FUNCTION_BLOCK FB_TrackSegment_1 EXTENDS FB_TrackBase IMPLEMENTS I_TRACK
VAR_INPUT
END_VAR
VAR_OUTPUT
END_VAR

METHOD Initialize : BOOL
VAR_INPUT
	nTrackIndex : UDINT;
END_VAR

VAR_INST
	TrackTable		: FB_TrackTable;
	
	nPointIndex		: INT;
	nPointIndexA	: INT;	
	nPointIndexB	: INT;	
	idx1, idx2		: INT;
	nStartFromTrack	: INT;
	nEndAtTrack		: INT;
	bCloseLoop		: BOOL;	
	
	bTrackBuild		: BOOL;
	StartFromTrack	: I_Track;
	EndAtTrack		: I_Track;
	
	sIndexWhereTheCheckFailed	: UINT;
	nErrorID					: UDINT;

END_VAR





VAR_INST
	
	TrackTableTemp		: ARRAY[1..gc_MaxNumberTrackPoints] OF ST_TrackTable;
	


END_VAR


VAR_INST
	
	pos01	:		PositionXYC;
	pos02	:		PositionXYC;


END_VAR

	  
CASE nState OF 

	10:	// Starting with an empty table. 
		IF TrackTable.ClearTrackTable() THEN
			nState := nState + 10;
		END_IF
		

	20:	// Init Track-Table
		
		// *************************************************************************************
		// *** Only the code in this state must be eddited according to machine/track layout ***
		// *************************************************************************************	
		
		nStartFromTrack	:= 0;		// 0 for the first track all others according to their predecessor!
	    	nEndAtTrack := 0;		// 0 for the first track all others according to their successor! 		
		     bCloseLoop := FALSE;	// TRUE for circular track	

			 			 			 
		// Building the track table:	
		TrackTable.AddPoint(E_PointType.Line_Start, E_PointOption.none, 480.0, 120.0, 0.0); 	 
		TrackTable.AddPoint(E_PointType.Line_End,   E_PointOption.none, 240.0, 120.0, 0.0);				
		
		TrackTable.AddPoint(E_PointType.Line_Start, E_PointOption.none, 120.0, 240.0, 0.0); 	 
		TrackTable.AddPoint(E_PointType.Line_End,   E_PointOption.none, 120.0, 480.0, 0.0);	
 
		TrackTable.AddPoint(E_PointType.Line_Start, E_PointOption.none, 240.0, 600.0, 0.0); 	 
		TrackTable.AddPoint(E_PointType.Line_End,   E_PointOption.none, 480.0, 600.0, 0.0);		
	 		
		nState := nState + 10;


	30:
		// *************************************************************
		// ***       NO Code Changes are needed from here on!        ***
		// *************************************************************		
			
		// The track table contains all additional information, too.
		IF nStartFromTrack > 0 THEN
			TrackTable.P_StartFromTrack := ipTrack[nStartFromTrack].std;	
		END_IF
		IF nEndAtTrack > 0 THEN
			TrackTable.P_EndAtTrack := ipTrack[nEndAtTrack].std;	
		END_IF	
		TrackTable.P_CloseTheLoop := bCloseLoop;	
		nState := nState + 10;

			
		
	40: // Checking the track table for plausibility
		IF TrackTable.CheckTrackTable() <> 0 THEN
			IF TrackTable.P_TrackTableCheckResult THEN
				nState := 50;	// Plausibility test succeeded.
			ELSE
				nState := 41;	// Plausibility test failed!
			END_IF
		END_IF

	
	41:	// In case of failed plausibility test check the creation of the above track table.
		// A Line must always begin with E_PointType.Line_Start and end with E_PointType.Line_End.
		// A Circle must always be added in the order E_PointType.Circle_Start, E_PointType.Circle_Center, E_PointType.Circle_End.
		// Check the info text for further information:
		sErrorInfoTextTemp := CONCAT('Track: ', UDINT_TO_STRING(nTrackIndex));
		sErrorInfoTextTemp := CONCAT(sErrorInfoTextTemp, ' - ');
		sErrorInfoTextTemp := CONCAT(sErrorInfoTextTemp, TrackTable.P_InfoText);
		
				     bTrackBuildError := TRUE;
					   sErrorInfoText := sErrorInfoTextTemp;
			sIndexWhereTheCheckFailed := TrackTable.P_TrackCheckImplausibleTableIndex;
					   TrackTableTemp := TrackTable.P_Table;	
							
 					   
	50:	// Building the track	
		IF fbTrackStandard.BuildTrackExt(TrackTable) THEN
			nState := nState +1;
		END_IF
		
	51:	IF fbTrackStandard.P_BuildTrackExt.Done THEN
			nState := 100;	
		ELSIF fbTrackStandard.P_BuildTrackExt.Error THEN
	  		nState := nState +1;
		END_IF		
		
	52: // In case an error occured, check the error ID and InfoText and react accordingly:
		sErrorInfoTextTemp := CONCAT('Track: ', UDINT_TO_STRING(nTrackIndex));
		sErrorInfoTextTemp := CONCAT(sErrorInfoTextTemp, ' - ');
		sErrorInfoTextTemp := CONCAT(sErrorInfoTextTemp, fbTrackStandard.P_BuildTrackExtInfoText);	
	
			      nErrorID := fbTrackStandard.P_BuildTrackExt.ErrorID;
		    sErrorInfoText := sErrorInfoTextTemp;		
			
		  bTrackBuildError := TRUE;		   
					   
		 
	100: 	// Track build done
			fTrackLength := fbTrackStandard.GetLength();
			  Initialize := TRUE;
	

END_CASE
END_METHOD

PROPERTY P_Error : BOOL
GET
P_Error := bTrackBuildError;
END_GET
END_PROPERTY

PROPERTY P_ErrorInfo : STRING
GET
P_ErrorInfo := sErrorInfoText;
END_GET
END_PROPERTY

END_FUNCTION_BLOCK

(* stored: Version 1.1.0.1, ProductVersion 3.1.4024.13
   POU FB_TrackSegment_1: Id {8bc03b03-a8a0-4837-bf56-60fab90a5b15}, SpecialFunc None
   Method Initialize: Id {ec4a5bb1-839f-4f43-b542-fc56fd640856}
   Property P_Error: Id {d386063a-b1d4-4b3c-940b-ef6404cff1d0}
   Get Get: Id {e4cd3f32-fa4c-420e-b6e4-48cb575ffb24}
   Property P_ErrorInfo: Id {1e4f03d0-c460-49e5-9817-32cb648de575}
   Get Get: Id {cb18e2b1-11c4-4a6d-abb3-214850a91257} *)
